FUNCTION_BLOCK BoolBindingReadOnlyTest EXTENDS TcUnit.FB_TestSuite
VAR
END_VAR

CheckIsBound();
BindingReturnsSameValue();
NegatedBindingReturnsNegatedValue();

METHOD BindingReturnsSameValue : BOOL
VAR
	expected : BOOL;
	actual : BOOL;
	
	binding : BoolBindingReadOnly;
	variable : BOOL;
END_VAR
TcUnit.TEST('Binding returns same value');

binding.Bind(variable);

expected := FALSE;
actual := binding.Value;

AssertEquals(
	Expected := expected,
	Actual := actual,
	Message := 'Value should return FALSE if bound variable is FALSE');
	
variable := TRUE;

expected := TRUE;
actual := binding.Value;

AssertEquals(
	Expected := expected,
	Actual := actual,
	Message := 'Value should return TRUE if bound variable is TRUE');

TEST_FINISHED();
END_METHOD

METHOD CheckIsBound : BOOL
VAR
	expected : BOOL;
	actual : BOOL;
	
	binding : BoolBindingReadOnly;
	variable : BOOL;
END_VAR
TcUnit.TEST('Check bound');

expected := FALSE;
actual := binding.IsBound;

AssertEquals(
	Expected := expected,
	Actual := actual,
	Message := 'IsBound should be FALSE before binding');

binding.Bind(variable);

expected := TRUE;
actual := binding.IsBound;

AssertEquals(
	Expected := expected,
	Actual := actual,
	Message := 'IsBound should be TRUE after successful Bind()');

TEST_FINISHED();
END_METHOD

METHOD NegatedBindingReturnsNegatedValue : BOOL
VAR
	expected : BOOL;
	actual : BOOL;
	
	binding : BoolBindingReadOnly;
	variable : BOOL;
END_VAR
TcUnit.TEST('Negated binding returns negated value');

binding.Bind(variable);
binding.Negate := TRUE;

expected := TRUE;
actual := binding.Value;

AssertEquals(
	Expected := expected,
	Actual := actual,
	Message := 'Value should return TRUE if bound variable is FALSE');
	
variable := TRUE;

expected := FALSE;
actual := binding.Value;

AssertEquals(
	Expected := expected,
	Actual := actual,
	Message := 'Value should return FALSE if bound variable is TRUE');

TEST_FINISHED();
END_METHOD

END_FUNCTION_BLOCK

(* stored: Version 1.1.0.1, ProductVersion 3.1.4024.15
   POU BoolBindingReadOnlyTest: Id {6f6aa6ee-3f80-0569-2a76-15890d9b574f}, SpecialFunc None
   Method BindingReturnsSameValue: Id {cf4f47ce-8a76-03d9-3c3a-c49c5b7d75ad}
   Method CheckIsBound: Id {20dbe522-faf1-0fc5-0fe6-786020207073}
   Method NegatedBindingReturnsNegatedValue: Id {3c48ae1d-44e9-0387-3f0c-4ea4ae8a5cfa} *)
